# EPICS autosave request: autosave/galil_forward_transform.req
$(P)$(M)_FTRANSFORM_SP
